# EPICS substitutions: viocs/si_ps/si_psApp/Db/kickers.substitutions
file "db/kickers.db" {
    pattern { family, pos }
        { "InjDK",  "01SA" }
        { "InjNLK", "01SA"}
}
